(* PLC project Untitled1, Beckhoff Automation GmbH TF6420 Database Server Query Analyser 1.0.0.0 *)
(* stored: creationDateTime 2024-01-05T13:26:19, modificationDateTime 2024-01-05T13:26:19 *)

TYPE ST_SelectStruct : STRUCT
  id : LINT;
  time2 : REAL;
  primary_power : REAL;
  secondary_power : REAL;
  phase_shift : REAL;
  frequency : REAL;
  flux_density : REAL;
  Meta_id : LINT;
END_STRUCT;
END_TYPE
